// TIA Portal V17 export
// export: Created 2021-12-03T08:13:10.1255312Z, ExportSetting WithDefaults, DisplayName Totally Integrated Automation Portal, DisplayVersion V17, DisplayName TIA Portal Openness, DisplayVersion V17, DisplayName TIA Portal Version Control Interface, DisplayVersion V17, DisplayName STEP 7 Professional, DisplayVersion V17, DisplayName STEP 7 Safety, DisplayVersion V17, DisplayName WinCC Advanced, DisplayVersion V17
DATA_BLOCK "FGDB_fCycle_Glob"   // DB3000, F_DB
VERSION : 0.1
// stored: AutoNumber false
   VAR
      AlwaysFalse : Bool;
      AlwaysTrue : Bool;
      AckCom : Bool;
   END_VAR
BEGIN
END_DATA_BLOCK
